	UF : 1, UT : 4,		CONFIG : 'N U T, 0, 0, 0',
	X =  145.000  mm,	Y =  154.000  mm,	Z =   15.000 mm,
	W =-180.000 deg,	P =   0.000 deg,	R =    90.000 deg
};
P[7454]{
   GP1:
	UF : 1, UT : 4,		CONFIG : 'N U T, 0, 0, 0',
	X =  145.000  mm,	Y =  154.000  mm,	Z =   -1.000 mm,
	W =-180.000 deg,	P =   0.000 deg,	R =    90.000 deg
};
P[7455]{
   GP1:
	UF : 1, UT : 4,		CONFIG : 'N U T, 0, 0, 0',
	X =  145.000  mm,	Y =  154.000  mm,	Z =   15.000 mm,
	W =-180.000 deg,	P =   0.000 deg,	R =    90.000 deg
};
P[7456]{
   GP1:
	UF : 1, UT : 4,		CONFIG : 'N U T, 0, 0, 0',
	X =  148.000  mm,	Y =  154.000  mm,	Z =   15.000 mm,
	W =-180.000 deg,	P =   0.000 deg,	R =    90.000 deg
};
P[7457]{
   GP1:
	UF : 1, UT : 4,		CONFIG : 'N U T, 0, 0, 0',
	X =  148.000  mm,	Y =  154.000  mm,	Z =   -1.000 mm,
	W =-180.000 deg,	P =   0.000 deg,	R =    90.000 deg
};
P[7458]{
   GP1:
	UF : 1, UT : 4,		CONFIG : 'N U T, 0, 0, 0',
	X =  148.000  mm,	Y =  154.000  mm,	Z =   15.000 mm,
	W =-180.000 deg,	P =   0.000 deg,	R =    90.000 deg
};
P[7459]{
   GP1:
	UF : 1, UT : 4,		CONFIG : 'N U T, 0, 0, 0',
	X =  151.000  mm,	Y =  154.000  mm,	Z =   15.000 mm,
	W =-180.000 deg,	P =   0.000 deg,	R =    90.000 deg
};
P[7460]{
   GP1:
	UF : 1, UT : 4,		CONFIG : 'N U T, 0, 0, 0',
	X =  151.000  mm,	Y =  154.000  mm,	Z =   -1.000 mm,
	W =-180.000 deg,	P =   0.000 deg,	R =    90.000 deg
};
P[7461]{
   GP1:
	UF : 1, UT : 4,		CONFIG : 'N U T, 0, 0, 0',
	X =  151.000  mm,	Y =  154.000  mm,	Z =   15.000 mm,
	W =-180.000 deg,	P =   0.000 deg,	R =    90.000 deg
};
P[7462]{
   GP1:
	UF : 1, UT : 4,		CONFIG : 'N U T, 0, 0, 0',
	X =  154.000  mm,	Y =  154.000  mm,	Z =   15.000 mm,
	W =-180.000 deg,	P =   0.000 deg,	R =    90.000 deg
};
P[7463]{
   GP1:
	UF : 1, UT : 4,		CONFIG : 'N U T, 0, 0, 0',
	X =  154.000  mm,	Y =  154.000  mm,	Z =   -1.000 mm,
	W =-180.000 deg,	P =   0.000 deg,	R =    90.000 deg
};
P[7464]{
   GP1:
	UF : 1, UT : 4,		CONFIG : 'N U T, 0, 0, 0',
	X =  154.000  mm,	Y =  154.000  mm,	Z =   15.000 mm,
	W =-180.000 deg,	P =   0.000 deg,	R =    90.000 deg
};
P[7474]{
   GP1:
	UF : 1, UT : 4,		CONFIG : 'N U T, 0, 0, 0',
	X =  25.000  mm,	Y =  157.000  mm,	Z =   15.000 mm,
	W =-180.000 deg,	P =   0.000 deg,	R =    90.000 deg
};
P[7475]{
   GP1:
	UF : 1, UT : 4,		CONFIG : 'N U T, 0, 0, 0',
	X =  25.000  mm,	Y =  157.000  mm,	Z =   -1.000 mm,
	W =-180.000 deg,	P =   0.000 deg,	R =    90.000 deg
};
P[7476]{
   GP1:
	UF : 1, UT : 4,		CONFIG : 'N U T, 0, 0, 0',
	X =  25.000  mm,	Y =  157.000  mm,	Z =   15.000 mm,
	W =-180.000 deg,	P =   0.000 deg,	R =    90.000 deg
};
P[7477]{
   GP1:
	UF : 1, UT : 4,		CONFIG : 'N U T, 0, 0, 0',
	X =  28.000  mm,	Y =  157.000  mm,	Z =   15.000 mm,
	W =-180.000 deg,	P =   0.000 deg,	R =    90.000 deg
};
P[7478]{
   GP1:
	UF : 1, UT : 4,		CONFIG : 'N U T, 0, 0, 0',
	X =  28.000  mm,	Y =  157.000  mm,	Z =   -1.000 mm,
	W =-180.000 deg,	P =   0.000 deg,	R =    90.000 deg
};
P[7479]{
   GP1:
	UF : 1, UT : 4,		CONFIG : 'N U T, 0, 0, 0',
	X =  28.000  mm,	Y =  157.000  mm,	Z =   15.000 mm,
	W =-180.000 deg,	P =   0.000 deg,	R =    90.000 deg
};
P[7480]{
   GP1:
	UF : 1, UT : 4,		CONFIG : 'N U T, 0, 0, 0',
	X =  31.000  mm,	Y =  157.000  mm,	Z =   15.000 mm,
	W =-180.000 deg,	P =   0.000 deg,	R =    90.000 deg
};
P[7481]{
   GP1:
	UF : 1, UT : 4,		CONFIG : 'N U T, 0, 0, 0',
	X =  31.000  mm,	Y =  157.000  mm,	Z =   -1.000 mm,
	W =-180.000 deg,	P =   0.000 deg,	R =    90.000 deg
};
P[7482]{
   GP1:
	UF : 1, UT : 4,		CONFIG : 'N U T, 0, 0, 0',
	X =  31.000  mm,	Y =  157.000  mm,	Z =   15.000 mm,
	W =-180.000 deg,	P =   0.000 deg,	R =    90.000 deg
};
P[7483]{
   GP1:
	UF : 1, UT : 4,		CONFIG : 'N U T, 0, 0, 0',
	X =  34.000  mm,	Y =  157.000  mm,	Z =   15.000 mm,
	W =-180.000 deg,	P =   0.000 deg,	R =    90.000 deg
};
P[7484]{
   GP1:
	UF : 1, UT : 4,		CONFIG : 'N U T, 0, 0, 0',
	X =  34.000  mm,	Y =  157.000  mm,	Z =   -1.000 mm,
	W =-180.000 deg,	P =   0.000 deg,	R =    90.000 deg
};
P[7485]{
   GP1:
	UF : 1, UT : 4,		CONFIG : 'N U T, 0, 0, 0',
	X =  34.000  mm,	Y =  157.000  mm,	Z =   15.000 mm,
	W =-180.000 deg,	P =   0.000 deg,	R =    90.000 deg
};
P[7486]{
   GP1:
	UF : 1, UT : 4,		CONFIG : 'N U T, 0, 0, 0',
	X =  37.000  mm,	Y =  157.000  mm,	Z =   15.000 mm,
	W =-180.000 deg,	P =   0.000 deg,	R =    90.000 deg
};
P[7487]{
   GP1:
	UF : 1, UT : 4,		CONFIG : 'N U T, 0, 0, 0',
	X =  37.000  mm,	Y =  157.000  mm,	Z =   -1.000 mm,
	W =-180.000 deg,	P =   0.000 deg,	R =    90.000 deg
};
P[7488]{
   GP1:
	UF : 1, UT : 4,		CONFIG : 'N U T, 0, 0, 0',
	X =  37.000  mm,	Y =  157.000  mm,	Z =   15.000 mm,
	W =-180.000 deg,	P =   0.000 deg,	R =    90.000 deg
};
P[7489]{
   GP1:
	UF : 1, UT : 4,		CONFIG : 'N U T, 0, 0, 0',
	X =  40.000  mm,	Y =  157.000  mm,	Z =   15.000 mm,
	W =-180.000 deg,	P =   0.000 deg,	R =    90.000 deg
};
P[7490]{
   GP1:
	UF : 1, UT : 4,		CONFIG : 'N U T, 0, 0, 0',
	X =  40.000  mm,	Y =  157.000  mm,	Z =   -1.000 mm,
	W =-180.000 deg,	P =   0.000 deg,	R =    90.000 deg
};
P[7491]{
   GP1:
	UF : 1, UT : 4,		CONFIG : 'N U T, 0, 0, 0',
	X =  40.000  mm,	Y =  157.000  mm,	Z =   15.000 mm,
	W =-180.000 deg,	P =   0.000 deg,	R =    90.000 deg
};
P[7492]{
   GP1:
	UF : 1, UT : 4,		CONFIG : 'N U T, 0, 0, 0',
	X =  43.000  mm,	Y =  157.000  mm,	Z =   15.000 mm,
	W =-180.000 deg,	P =   0.000 deg,	R =    90.000 deg
};
P[7493]{
   GP1:
	UF : 1, UT : 4,		CONFIG : 'N U T, 0, 0, 0',
	X =  43.000  mm,	Y =  157.000  mm,	Z =   -1.000 mm,
	W =-180.000 deg,	P =   0.000 deg,	R =    90.000 deg
};
P[7494]{
   GP1:
	UF : 1, UT : 4,		CONFIG : 'N U T, 0, 0, 0',
	X =  43.000  mm,	Y =  157.000  mm,	Z =   15.000 mm,
	W =-180.000 deg,	P =   0.000 deg,	R =    90.000 deg
};
P[7495]{
   GP1:
	UF : 1, UT : 4,		CONFIG : 'N U T, 0, 0, 0',
	X =  46.000  mm,	Y =  157.000  mm,	Z =   15.000 mm,
	W =-180.000 deg,	P =   0.000 deg,	R =    90.000 deg
};
P[7496]{
   GP1:
	UF : 1, UT : 4,		CONFIG : 'N U T, 0, 0, 0',
	X =  46.000  mm,	Y =  157.000  mm,	Z =   -1.000 mm,
	W =-180.000 deg,	P =   0.000 deg,	R =    90.000 deg
};
P[7497]{
   GP1:
	UF : 1, UT : 4,		CONFIG : 'N U T, 0, 0, 0',
	X =  46.000  mm,	Y =  157.000  mm,	Z =   15.000 mm,
	W =-180.000 deg,	P =   0.000 deg,	R =    90.000 deg
};
P[7498]{
   GP1:
	UF : 1, UT : 4,		CONFIG : 'N U T, 0, 0, 0',
	X =  49.000  mm,	Y =  157.000  mm,	Z =   15.000 mm,
	W =-180.000 deg,	P =   0.000 deg,	R =    90.000 deg
};
P[7499]{
   GP1:
	UF : 1, UT : 4,		CONFIG : 'N U T, 0, 0, 0',
	X =  49.000  mm,	Y =  157.000  mm,	Z =   -1.000 mm,
	W =-180.000 deg,	P =   0.000 deg,	R =    90.000 deg
};
P[7500]{
   GP1:
	UF : 1, UT : 4,		CONFIG : 'N U T, 0, 0, 0',
	X =  49.000  mm,	Y =  157.000  mm,	Z =   15.000 mm,
	W =-180.000 deg,	P =   0.000 deg,	R =    90.000 deg
};
P[7501]{
   GP1:
	UF : 1, UT : 4,		CONFIG : 'N U T, 0, 0, 0',
	X =  52.000  mm,	Y =  157.000  mm,	Z =   15.000 mm,
	W =-180.000 deg,	P =   0.000 deg,	R =    90.000 deg
};
P[7502]{
   GP1:
	UF : 1, UT : 4,		CONFIG : 'N U T, 0, 0, 0',
	X =  52.000  mm,	Y =  157.000  mm,	Z =   -1.000 mm,
	W =-180.000 deg,	P =   0.000 deg,	R =    90.000 deg
};
P[7503]{
   GP1:
	UF : 1, UT : 4,		CONFIG : 'N U T, 0, 0, 0',
	X =  52.000  mm,	Y =  157.000  mm,	Z =   15.000 mm,
	W =-180.000 deg,	P =   0.000 deg,	R =    90.000 deg
};
P[7504]{
   GP1:
	UF : 1, UT : 4,		CONFIG : 'N U T, 0, 0, 0',
	X =  55.000  mm,	Y =  157.000  mm,	Z =   15.000 mm,
	W =-180.000 deg,	P =   0.000 deg,	R =    90.000 deg
};
P[7505]{
   GP1:
	UF : 1, UT : 4,		CONFIG : 'N U T, 0, 0, 0',
	X =  55.000  mm,	Y =  157.000  mm,	Z =   -1.000 mm,
	W =-180.000 deg,	P =   0.000 deg,	R =    90.000 deg
};
P[7506]{
   GP1:
	UF : 1, UT : 4,		CONFIG : 'N U T, 0, 0, 0',
	X =  55.000  mm,	Y =  157.000  mm,	Z =   15.000 mm,
	W =-180.000 deg,	P =   0.000 deg,	R =    90.000 deg
};
P[7507]{
   GP1:
	UF : 1, UT : 4,		CONFIG : 'N U T, 0, 0, 0',
	X =  58.000  mm,	Y =  157.000  mm,	Z =   15.000 mm,
	W =-180.000 deg,	P =   0.000 deg,	R =    90.000 deg
};
P[7508]{
   GP1:
	UF : 1, UT : 4,		CONFIG : 'N U T, 0, 0, 0',
	X =  58.000  mm,	Y =  157.000  mm,	Z =   -1.000 mm,
	W =-180.000 deg,	P =   0.000 deg,	R =    90.000 deg
};
P[7509]{
   GP1:
	UF : 1, UT : 4,		CONFIG : 'N U T, 0, 0, 0',
	X =  58.000  mm,	Y =  157.000  mm,	Z =   15.000 mm,
	W =-180.000 deg,	P =   0.000 deg,	R =    90.000 deg
};
P[7516]{
   GP1:
	UF : 1, UT : 4,		CONFIG : 'N U T, 0, 0, 0',
	X =  109.000  mm,	Y =  157.000  mm,	Z =   15.000 mm,
	W =-180.000 deg,	P =   0.000 deg,	R =    90.000 deg
};
P[7517]{
   GP1:
	UF : 1, UT : 4,		CONFIG : 'N U T, 0, 0, 0',
	X =  109.000  mm,	Y =  157.000  mm,	Z =   -1.000 mm,
	W =-180.000 deg,	P =   0.000 deg,	R =    90.000 deg
};
P[7518]{
   GP1:
	UF : 1, UT : 4,		CONFIG : 'N U T, 0, 0, 0',
	X =  109.000  mm,	Y =  157.000  mm,	Z =   15.000 mm,
	W =-180.000 deg,	P =   0.000 deg,	R =    90.000 deg
};
P[7549]{
   GP1:
	UF : 1, UT : 4,		CONFIG : 'N U T, 0, 0, 0',
	X =  142.000  mm,	Y =  157.000  mm,	Z =   15.000 mm,
	W =-180.000 deg,	P =   0.000 deg,	R =    90.000 deg
};
P[7550]{
   GP1:
	UF : 1, UT : 4,		CONFIG : 'N U T, 0, 0, 0',
	X =  142.000  mm,	Y =  157.000  mm,	Z =   -1.000 mm,
	W =-180.000 deg,	P =   0.000 deg,	R =    90.000 deg
};
P[7551]{
   GP1:
	UF : 1, UT : 4,		CONFIG : 'N U T, 0, 0, 0',
	X =  142.000  mm,	Y =  157.000  mm,	Z =   15.000 mm,
	W =-180.000 deg,	P =   0.000 deg,	R =    90.000 deg
};
P[7552]{
   GP1:
	UF : 1, UT : 4,		CONFIG : 'N U T, 0, 0, 0',
	X =  145.000  mm,	Y =  157.000  mm,	Z =   15.000 mm,
	W =-180.000 deg,	P =   0.000 deg,	R =    90.000 deg
};
P[7553]{
   GP1:
	UF : 1, UT : 4,		CONFIG : 'N U T, 0, 0, 0',
	X =  145.000  mm,	Y =  157.000  mm,	Z =   -1.000 mm,
	W =-180.000 deg,	P =   0.000 deg,	R =    90.000 deg
};
P[7554]{
   GP1:
	UF : 1, UT : 4,		CONFIG : 'N U T, 0, 0, 0',
	X =  145.000  mm,	Y =  157.000  mm,	Z =   15.000 mm,
	W =-180.000 deg,	P =   0.000 deg,	R =    90.000 deg
};
P[7555]{
   GP1:
	UF : 1, UT : 4,		CONFIG : 'N U T, 0, 0, 0',
	X =  148.000  mm,	Y =  157.000  mm,	Z =   15.000 mm,
	W =-180.000 deg,	P =   0.000 deg,	R =    90.000 deg
};
P[7556]{
   GP1:
	UF : 1, UT : 4,		CONFIG : 'N U T, 0, 0, 0',
	X =  148.000  mm,	Y =  157.000  mm,	Z =   -1.000 mm,
	W =-180.000 deg,	P =   0.000 deg,	R =    90.000 deg
};
P[7557]{
   GP1:
	UF : 1, UT : 4,		CONFIG : 'N U T, 0, 0, 0',
	X =  148.000  mm,	Y =  157.000  mm,	Z =   15.000 mm,
	W =-180.000 deg,	P =   0.000 deg,	R =    90.000 deg
};
P[7558]{
   GP1:
	UF : 1, UT : 4,		CONFIG : 'N U T, 0, 0, 0',
	X =  151.000  mm,	Y =  157.000  mm,	Z =   15.000 mm,
	W =-180.000 deg,	P =   0.000 deg,	R =    90.000 deg
};
P[7559]{
   GP1:
	UF : 1, UT : 4,		CONFIG : 'N U T, 0, 0, 0',
	X =  151.000  mm,	Y =  157.000  mm,	Z =   -1.000 mm,
	W =-180.000 deg,	P =   0.000 deg,	R =    90.000 deg
};
P[7560]{
   GP1:
	UF : 1, UT : 4,		CONFIG : 'N U T, 0, 0, 0',
	X =  151.000  mm,	Y =  157.000  mm,	Z =   15.000 mm,
	W =-180.000 deg,	P =   0.000 deg,	R =    90.000 deg
};
P[7561]{
   GP1:
	UF : 1, UT : 4,		CONFIG : 'N U T, 0, 0, 0',
	X =  154.000  mm,	Y =  157.000  mm,	Z =   15.000 mm,
	W =-180.000 deg,	P =   0.000 deg,	R =    90.000 deg
};
P[7562]{
   GP1:
	UF : 1, UT : 4,		CONFIG : 'N U T, 0, 0, 0',
	X =  154.000  mm,	Y =  157.000  mm,	Z =   -1.000 mm,
	W =-180.000 deg,	P =   0.000 deg,	R =    90.000 deg
};
P[7563]{
   GP1:
	UF : 1, UT : 4,		CONFIG : 'N U T, 0, 0, 0',
	X =  154.000  mm,	Y =  157.000  mm,	Z =   15.000 mm,
	W =-180.000 deg,	P =   0.000 deg,	R =    90.000 deg
};
P[7615]{
   GP1:
	UF : 1, UT : 4,		CONFIG : 'N U T, 0, 0, 0',
	X =  109.000  mm,	Y =  160.000  mm,	Z =   15.000 mm,
	W =-180.000 deg,	P =   0.000 deg,	R =    90.000 deg
};
P[7616]{
   GP1:
	UF : 1, UT : 4,		CONFIG : 'N U T, 0, 0, 0',
	X =  109.000  mm,	Y =  160.000  mm,	Z =   -1.000 mm,
	W =-180.000 deg,	P =   0.000 deg,	R =    90.000 deg
};
P[7617]{
   GP1:
	UF : 1, UT : 4,		CONFIG : 'N U T, 0, 0, 0',
	X =  109.000  mm,	Y =  160.000  mm,	Z =   15.000 mm,
	W =-180.000 deg,	P =   0.000 deg,	R =    90.000 deg
};
P[7618]{
   GP1:
	UF : 1, UT : 4,		CONFIG : 'N U T, 0, 0, 0',
	X =  112.000  mm,	Y =  160.000  mm,	Z =   15.000 mm,
	W =-180.000 deg,	P =   0.000 deg,	R =    90.000 deg
};
P[7619]{
   GP1:
	UF : 1, UT : 4,		CONFIG : 'N U T, 0, 0, 0',
	X =  112.000  mm,	Y =  160.000  mm,	Z =   -1.000 mm,
	W =-180.000 deg,	P =   0.000 deg,	R =    90.000 deg
};
P[7620]{
   GP1:
	UF : 1, UT : 4,		CONFIG : 'N U T, 0, 0, 0',
	X =  112.000  mm,	Y =  160.000  mm,	Z =   15.000 mm,
	W =-180.000 deg,	P =   0.000 deg,	R =    90.000 deg
};
P[7651]{
   GP1:
	UF : 1, UT : 4,		CONFIG : 'N U T, 0, 0, 0',
	X =  145.000  mm,	Y =  160.000  mm,	Z =   15.000 mm,
	W =-180.000 deg,	P =   0.000 deg,	R =    90.000 deg
};
P[7652]{
   GP1:
	UF : 1, UT : 4,		CONFIG : 'N U T, 0, 0, 0',
	X =  145.000  mm,	Y =  160.000  mm,	Z =   -1.000 mm,
	W =-180.000 deg,	P =   0.000 deg,	R =    90.000 deg
};
P[7653]{
   GP1:
	UF : 1, UT : 4,		CONFIG : 'N U T, 0, 0, 0',
	X =  145.000  mm,	Y =  160.000  mm,	Z =   15.000 mm,
	W =-180.000 deg,	P =   0.000 deg,	R =    90.000 deg
};
P[7654]{
   GP1:
	UF : 1, UT : 4,		CONFIG : 'N U T, 0, 0, 0',
	X =  148.000  mm,	Y =  160.000  mm,	Z =   15.000 mm,
	W =-180.000 deg,	P =   0.000 deg,	R =    90.000 deg
};
P[7655]{
   GP1:
	UF : 1, UT : 4,		CONFIG : 'N U T, 0, 0, 0',
	X =  148.000  mm,	Y =  160.000  mm,	Z =   -1.000 mm,
	W =-180.000 deg,	P =   0.000 deg,	R =    90.000 deg
};
P[7656]{
   GP1:
	UF : 1, UT : 4,		CONFIG : 'N U T, 0, 0, 0',
	X =  148.000  mm,	Y =  160.000  mm,	Z =   15.000 mm,
	W =-180.000 deg,	P =   0.000 deg,	R =    90.000 deg
};
P[7663]{
   GP1:
	UF : 1, UT : 4,		CONFIG : 'N U T, 0, 0, 0',
	X =  22.000  mm,	Y =  163.000  mm,	Z =   15.000 mm,
	W =-180.000 deg,	P =   0.000 deg,	R =    90.000 deg
};
P[7664]{
   GP1:
	UF : 1, UT : 4,		CONFIG : 'N U T, 0, 0, 0',
	X =  22.000  mm,	Y =  163.000  mm,	Z =   -1.000 mm,
	W =-180.000 deg,	P =   0.000 deg,	R =    90.000 deg
};
P[7665]{
   GP1:
	UF : 1, UT : 4,		CONFIG : 'N U T, 0, 0, 0',
	X =  22.000  mm,	Y =  163.000  mm,	Z =   15.000 mm,
	W =-180.000 deg,	P =   0.000 deg,	R =    90.000 deg
};
P[7708]{
   GP1:
	UF : 1, UT : 4,		CONFIG : 'N U T, 0, 0, 0',
	X =  109.000  mm,	Y =  163.000  mm,	Z =   15.000 mm,
	W =-180.000 deg,	P =   0.000 deg,	R =    90.000 deg
};
P[7709]{
   GP1:
	UF : 1, UT : 4,		CONFIG : 'N U T, 0, 0, 0',
	X =  109.000  mm,	Y =  163.000  mm,	Z =   -1.000 mm,
	W =-180.000 deg,	P =   0.000 deg,	R =    90.000 deg
};
P[7710]{
   GP1:
	UF : 1, UT : 4,		CONFIG : 'N U T, 0, 0, 0',
	X =  109.000  mm,	Y =  163.000  mm,	Z =   15.000 mm,
	W =-180.000 deg,	P =   0.000 deg,	R =    90.000 deg
};
P[7711]{
   GP1:
	UF : 1, UT : 4,		CONFIG : 'N U T, 0, 0, 0',
	X =  112.000  mm,	Y =  163.000  mm,	Z =   15.000 mm,
	W =-180.000 deg,	P =   0.000 deg,	R =    90.000 deg
};
P[7712]{
   GP1:
	UF : 1, UT : 4,		CONFIG : 'N U T, 0, 0, 0',
	X =  112.000  mm,	Y =  163.000  mm,	Z =   -1.000 mm,
	W =-180.000 deg,	P =   0.000 deg,	R =    90.000 deg
};
P[7713]{
   GP1:
	UF : 1, UT : 4,		CONFIG : 'N U T, 0, 0, 0',
	X =  112.000  mm,	Y =  163.000  mm,	Z =   15.000 mm,
	W =-180.000 deg,	P =   0.000 deg,	R =    90.000 deg
};
P[7720]{
   GP1:
	UF : 1, UT : 4,		CONFIG : 'N U T, 0, 0, 0',
	X =  121.000  mm,	Y =  163.000  mm,	Z =   15.000 mm,
	W =-180.000 deg,	P =   0.000 deg,	R =    90.000 deg
};
P[7721]{
   GP1:
	UF : 1, UT : 4,		CONFIG : 'N U T, 0, 0, 0',
	X =  121.000  mm,	Y =  163.000  mm,	Z =   -1.000 mm,
	W =-180.000 deg,	P =   0.000 deg,	R =    90.000 deg
};
P[7722]{
   GP1:
	UF : 1, UT : 4,		CONFIG : 'N U T, 0, 0, 0',
	X =  121.000  mm,	Y =  163.000  mm,	Z =   15.000 mm,
	W =-180.000 deg,	P =   0.000 deg,	R =    90.000 deg
};
P[7723]{
   GP1:
	UF : 1, UT : 4,		CONFIG : 'N U T, 0, 0, 0',
	X =  124.000  mm,	Y =  163.000  mm,	Z =   15.000 mm,
	W =-180.000 deg,	P =   0.000 deg,	R =    90.000 deg
};
P[7724]{
   GP1:
	UF : 1, UT : 4,		CONFIG : 'N U T, 0, 0, 0',
	X =  124.000  mm,	Y =  163.000  mm,	Z =   -1.000 mm,
	W =-180.000 deg,	P =   0.000 deg,	R =    90.000 deg
};
P[7725]{
   GP1:
	UF : 1, UT : 4,		CONFIG : 'N U T, 0, 0, 0',
	X =  124.000  mm,	Y =  163.000  mm,	Z =   15.000 mm,
	W =-180.000 deg,	P =   0.000 deg,	R =    90.000 deg
};
P[7726]{
   GP1:
	UF : 1, UT : 4,		CONFIG : 'N U T, 0, 0, 0',
	X =  127.000  mm,	Y =  163.000  mm,	Z =   15.000 mm,
	W =-180.000 deg,	P =   0.000 deg,	R =    90.000 deg
};
P[7727]{
   GP1:
	UF : 1, UT : 4,		CONFIG : 'N U T, 0, 0, 0',
	X =  127.000  mm,	Y =  163.000  mm,	Z =   -1.000 mm,
	W =-180.000 deg,	P =   0.000 deg,	R =    90.000 deg
};
P[7728]{
   GP1:
	UF : 1, UT : 4,		CONFIG : 'N U T, 0, 0, 0',
	X =  127.000  mm,	Y =  163.000  mm,	Z =   15.000 mm,
	W =-180.000 deg,	P =   0.000 deg,	R =    90.000 deg
};
P[7729]{
   GP1:
	UF : 1, UT : 4,		CONFIG : 'N U T, 0, 0, 0',
	X =  130.000  mm,	Y =  163.000  mm,	Z =   15.000 mm,
	W =-180.000 deg,	P =   0.000 deg,	R =    90.000 deg
};
P[7730]{
   GP1:
	UF : 1, UT : 4,		CONFIG : 'N U T, 0, 0, 0',
	X =  130.000  mm,	Y =  163.000  mm,	Z =   -1.000 mm,
	W =-180.000 deg,	P =   0.000 deg,	R =    90.000 deg
};
P[7731]{
   GP1:
	UF : 1, UT : 4,		CONFIG : 'N U T, 0, 0, 0',
	X =  130.000  mm,	Y =  163.000  mm,	Z =   15.000 mm,
	W =-180.000 deg,	P =   0.000 deg,	R =    90.000 deg
};
P[7732]{
   GP1:
	UF : 1, UT : 4,		CONFIG : 'N U T, 0, 0, 0',
	X =  133.000  mm,	Y =  163.000  mm,	Z =   15.000 mm,
	W =-180.000 deg,	P =   0.000 deg,	R =    90.000 deg
};
P[7733]{
   GP1:
	UF : 1, UT : 4,		CONFIG : 'N U T, 0, 0, 0',
	X =  133.000  mm,	Y =  163.000  mm,	Z =   -1.000 mm,
	W =-180.000 deg,	P =   0.000 deg,	R =    90.000 deg
};
P[7734]{
   GP1:
	UF : 1, UT : 4,		CONFIG : 'N U T, 0, 0, 0',
	X =  133.000  mm,	Y =  163.000  mm,	Z =   15.000 mm,
	W =-180.000 deg,	P =   0.000 deg,	R =    90.000 deg
};
P[7735]{
   GP1:
	UF : 1, UT : 4,		CONFIG : 'N U T, 0, 0, 0',
	X =  136.000  mm,	Y =  163.000  mm,	Z =   15.000 mm,
	W =-180.000 deg,	P =   0.000 deg,	R =    90.000 deg
};
P[7736]{
   GP1:
	UF : 1, UT : 4,		CONFIG : 'N U T, 0, 0, 0',
	X =  136.000  mm,	Y =  163.000  mm,	Z =   -1.000 mm,
	W =-180.000 deg,	P =   0.000 deg,	R =    90.000 deg
};
P[7737]{
   GP1:
	UF : 1, UT : 4,		CONFIG : 'N U T, 0, 0, 0',
	X =  136.000  mm,	Y =  163.000  mm,	Z =   15.000 mm,
	W =-180.000 deg,	P =   0.000 deg,	R =    90.000 deg
};
P[7738]{
   GP1:
	UF : 1, UT : 4,		CONFIG : 'N U T, 0, 0, 0',
	X =  139.000  mm,	Y =  163.000  mm,	Z =   15.000 mm,
	W =-180.000 deg,	P =   0.000 deg,	R =    90.000 deg
};
P[7739]{
   GP1:
	UF : 1, UT : 4,		CONFIG : 'N U T, 0, 0, 0',
	X =  139.000  mm,	Y =  163.000  mm,	Z =   -1.000 mm,
	W =-180.000 deg,	P =   0.000 deg,	R =    90.000 deg
};
P[7740]{
   GP1:
	UF : 1, UT : 4,		CONFIG : 'N U T, 0, 0, 0',
	X =  139.000  mm,	Y =  163.000  mm,	Z =   15.000 mm,
	W =-180.000 deg,	P =   0.000 deg,	R =    90.000 deg
};
P[7741]{
   GP1:
	UF : 1, UT : 4,		CONFIG : 'N U T, 0, 0, 0',
	X =  142.000  mm,	Y =  163.000  mm,	Z =   15.000 mm,
	W =-180.000 deg,	P =   0.000 deg,	R =    90.000 deg
};
P[7742]{
   GP1:
	UF : 1, UT : 4,		CONFIG : 'N U T, 0, 0, 0',
	X =  142.000  mm,	Y =  163.000  mm,	Z =   -1.000 mm,
	W =-180.000 deg,	P =   0.000 deg,	R =    90.000 deg
};
P[7743]{
   GP1:
	UF : 1, UT : 4,		CONFIG : 'N U T, 0, 0, 0',
	X =  142.000  mm,	Y =  163.000  mm,	Z =   15.000 mm,
	W =-180.000 deg,	P =   0.000 deg,	R =    90.000 deg
};
P[7744]{
   GP1:
	UF : 1, UT : 4,		CONFIG : 'N U T, 0, 0, 0',
	X =  145.000  mm,	Y =  163.000  mm,	Z =   15.000 mm,
	W =-180.000 deg,	P =   0.000 deg,	R =    90.000 deg
};
P[7745]{
   GP1:
	UF : 1, UT : 4,		CONFIG : 'N U T, 0, 0, 0',
	X =  145.000  mm,	Y =  163.000  mm,	Z =   -1.000 mm,
	W =-180.000 deg,	P =   0.000 deg,	R =    90.000 deg
};
P[7746]{
   GP1:
	UF : 1, UT : 4,		CONFIG : 'N U T, 0, 0, 0',
	X =  145.000  mm,	Y =  163.000  mm,	Z =   15.000 mm,
	W =-180.000 deg,	P =   0.000 deg,	R =    90.000 deg
};
P[7747]{
   GP1:
	UF : 1, UT : 4,		CONFIG : 'N U T, 0, 0, 0',
	X =  148.000  mm,	Y =  163.000  mm,	Z =   15.000 mm,
	W =-180.000 deg,	P =   0.000 deg,	R =    90.000 deg
};
P[7748]{
   GP1:
	UF : 1, UT : 4,		CONFIG : 'N U T, 0, 0, 0',
	X =  148.000  mm,	Y =  163.000  mm,	Z =   -1.000 mm,
	W =-180.000 deg,	P =   0.000 deg,	R =    90.000 deg
};
P[7749]{
   GP1:
	UF : 1, UT : 4,		CONFIG : 'N U T, 0, 0, 0',
	X =  148.000  mm,	Y =  163.000  mm,	Z =   15.000 mm,
	W =-180.000 deg,	P =   0.000 deg,	R =    90.000 deg
};
P[7780]{
   GP1:
	UF : 1, UT : 4,		CONFIG : 'N U T, 0, 0, 0',
	X =  49.000  mm,	Y =  166.000  mm,	Z =   15.000 mm,
	W =-180.000 deg,	P =   0.000 deg,	R =    90.000 deg
};
P[7781]{
   GP1:
	UF : 1, UT : 4,		CONFIG : 'N U T, 0, 0, 0',
	X =  49.000  mm,	Y =  166.000  mm,	Z =   -1.000 mm,
	W =-180.000 deg,	P =   0.000 deg,	R =    90.000 deg
};
P[7782]{
   GP1:
	UF : 1, UT : 4,		CONFIG : 'N U T, 0, 0, 0',
	X =  49.000  mm,	Y =  166.000  mm,	Z =   15.000 mm,
	W =-180.000 deg,	P =   0.000 deg,	R =    90.000 deg
};
P[7795]{
   GP1:
	UF : 1, UT : 4,		CONFIG : 'N U T, 0, 0, 0',
	X =  109.000  mm,	Y =  166.000  mm,	Z =   15.000 mm,
	W =-180.000 deg,	P =   0.000 deg,	R =    90.000 deg
};
P[7796]{
   GP1:
	UF : 1, UT : 4,		CONFIG : 'N U T, 0, 0, 0',
	X =  109.000  mm,	Y =  166.000  mm,	Z =   -1.000 mm,
	W =-180.000 deg,	P =   0.000 deg,	R =    90.000 deg
};
P[7797]{
   GP1:
	UF : 1, UT : 4,		CONFIG : 'N U T, 0, 0, 0',
	X =  109.000  mm,	Y =  166.000  mm,	Z =   15.000 mm,
	W =-180.000 deg,	P =   0.000 deg,	R =    90.000 deg
};
P[7798]{
   GP1:
	UF : 1, UT : 4,		CONFIG : 'N U T, 0, 0, 0',
	X =  112.000  mm,	Y =  166.000  mm,	Z =   15.000 mm,
	W =-180.000 deg,	P =   0.000 deg,	R =    90.000 deg
};
P[7799]{
   GP1:
	UF : 1, UT : 4,		CONFIG : 'N U T, 0, 0, 0',
	X =  112.000  mm,	Y =  166.000  mm,	Z =   -1.000 mm,
	W =-180.000 deg,	P =   0.000 deg,	R =    90.000 deg
};
P[7800]{
   GP1:
	UF : 1, UT : 4,		CONFIG : 'N U T, 0, 0, 0',
	X =  112.000  mm,	Y =  166.000  mm,	Z =   15.000 mm,
	W =-180.000 deg,	P =   0.000 deg,	R =    90.000 deg
};
P[7813]{
   GP1:
	UF : 1, UT : 4,		CONFIG : 'N U T, 0, 0, 0',
	X =  127.000  mm,	Y =  166.000  mm,	Z =   15.000 mm,
	W =-180.000 deg,	P =   0.000 deg,	R =    90.000 deg
};
P[7814]{
   GP1:
	UF : 1, UT : 4,		CONFIG : 'N U T, 0, 0, 0',
	X =  127.000  mm,	Y =  166.000  mm,	Z =   -1.000 mm,
	W =-180.000 deg,	P =   0.000 deg,	R =    90.000 deg
};
P[7815]{
   GP1:
	UF : 1, UT : 4,		CONFIG : 'N U T, 0, 0, 0',
	X =  127.000  mm,	Y =  166.000  mm,	Z =   15.000 mm,
	W =-180.000 deg,	P =   0.000 deg,	R =    90.000 deg
};
P[7816]{
   GP1:
	UF : 1, UT : 4,		CONFIG : 'N U T, 0, 0, 0',
	X =  130.000  mm,	Y =  166.000  mm,	Z =   15.000 mm,
	W =-180.000 deg,	P =   0.000 deg,	R =    90.000 deg
};
P[7817]{
   GP1:
	UF : 1, UT : 4,		CONFIG : 'N U T, 0, 0, 0',
	X =  130.000  mm,	Y =  166.000  mm,	Z =   -1.000 mm,
	W =-180.000 deg,	P =   0.000 deg,	R =    90.000 deg
};
P[7818]{
   GP1:
	UF : 1, UT : 4,		CONFIG : 'N U T, 0, 0, 0',
	X =  130.000  mm,	Y =  166.000  mm,	Z =   15.000 mm,
	W =-180.000 deg,	P =   0.000 deg,	R =    90.000 deg
};
P[7819]{
   GP1:
	UF : 1, UT : 4,		CONFIG : 'N U T, 0, 0, 0',
	X =  133.000  mm,	Y =  166.000  mm,	Z =   15.000 mm,
	W =-180.000 deg,	P =   0.000 deg,	R =    90.000 deg
};
P[7820]{
   GP1:
	UF : 1, UT : 4,		CONFIG : 'N U T, 0, 0, 0',
	X =  133.000  mm,	Y =  166.000  mm,	Z =   -1.000 mm,
	W =-180.000 deg,	P =   0.000 deg,	R =    90.000 deg
};
P[7821]{
   GP1:
	UF : 1, UT : 4,		CONFIG : 'N U T, 0, 0, 0',
	X =  133.000  mm,	Y =  166.000  mm,	Z =   15.000 mm,
	W =-180.000 deg,	P =   0.000 deg,	R =    90.000 deg
};
P[7822]{
   GP1:
	UF : 1, UT : 4,		CONFIG : 'N U T, 0, 0, 0',
	X =  136.000  mm,	Y =  166.000  mm,	Z =   15.000 mm,
	W =-180.000 deg,	P =   0.000 deg,	R =    90.000 deg
};
P[7823]{
   GP1:
	UF : 1, UT : 4,		CONFIG : 'N U T, 0, 0, 0',
	X =  136.000  mm,	Y =  166.000  mm,	Z =   -1.000 mm,
	W =-180.000 deg,	P =   0.000 deg,	R =    90.000 deg
};
P[7824]{
   GP1:
	UF : 1, UT : 4,		CONFIG : 'N U T, 0, 0, 0',
	X =  136.000  mm,	Y =  166.000  mm,	Z =   15.000 mm,
	W =-180.000 deg,	P =   0.000 deg,	R =    90.000 deg
};
P[7825]{
   GP1:
	UF : 1, UT : 4,		CONFIG : 'N U T, 0, 0, 0',
	X =  139.000  mm,	Y =  166.000  mm,	Z =   15.000 mm,
	W =-180.000 deg,	P =   0.000 deg,	R =    90.000 deg
};
P[7826]{
   GP1:
	UF : 1, UT : 4,		CONFIG : 'N U T, 0, 0, 0',
	X =  139.000  mm,	Y =  166.000  mm,	Z =   -1.000 mm,
	W =-180.000 deg,	P =   0.000 deg,	R =    90.000 deg
};
P[7827]{
   GP1:
	UF : 1, UT : 4,		CONFIG : 'N U T, 0, 0, 0',
	X =  139.000  mm,	Y =  166.000  mm,	Z =   15.000 mm,
	W =-180.000 deg,	P =   0.000 deg,	R =    90.000 deg
};
P[7828]{
   GP1:
	UF : 1, UT : 4,		CONFIG : 'N U T, 0, 0, 0',
	X =  142.000  mm,	Y =  166.000  mm,	Z =   15.000 mm,
	W =-180.000 deg,	P =   0.000 deg,	R =    90.000 deg
};
P[7829]{
   GP1:
	UF : 1, UT : 4,		CONFIG : 'N U T, 0, 0, 0',
	X =  142.000  mm,	Y =  166.000  mm,	Z =   -1.000 mm,
	W =-180.000 deg,	P =   0.000 deg,	R =    90.000 deg
};
P[7830]{
   GP1:
	UF : 1, UT : 4,		CONFIG : 'N U T, 0, 0, 0',
	X =  142.000  mm,	Y =  166.000  mm,	Z =   15.000 mm,
	W =-180.000 deg,	P =   0.000 deg,	R =    90.000 deg
};
P[7831]{
   GP1:
	UF : 1, UT : 4,		CONFIG : 'N U T, 0, 0, 0',
	X =  145.000  mm,	Y =  166.000  mm,	Z =   15.000 mm,
	W =-180.000 deg,	P =   0.000 deg,	R =    90.000 deg
};
P[7832]{
   GP1:
	UF : 1, UT : 4,		CONFIG : 'N U T, 0, 0, 0',
	X =  145.000  mm,	Y =  166.000  mm,	Z =   -1.000 mm,
	W =-180.000 deg,	P =   0.000 deg,	R =    90.000 deg
};
P[7833]{
   GP1:
	UF : 1, UT : 4,		CONFIG : 'N U T, 0, 0, 0',
	X =  145.000  mm,	Y =  166.000  mm,	Z =   15.000 mm,
	W =-180.000 deg,	P =   0.000 deg,	R =    90.000 deg
};
P[7834]{
   GP1:
	UF : 1, UT : 4,		CONFIG : 'N U T, 0, 0, 0',
	X =  148.000  mm,	Y =  166.000  mm,	Z =   15.000 mm,
	W =-180.000 deg,	P =   0.000 deg,	R =    90.000 deg
};
P[7835]{
   GP1:
	UF : 1, UT : 4,		CONFIG : 'N U T, 0, 0, 0',
	X =  148.000  mm,	Y =  166.000  mm,	Z =   -1.000 mm,
	W =-180.000 deg,	P =   0.000 deg,	R =    90.000 deg
};
P[7836]{
   GP1:
	UF : 1, UT : 4,		CONFIG : 'N U T, 0, 0, 0',
	X =  148.000  mm,	Y =  166.000  mm,	Z =   15.000 mm,
	W =-180.000 deg,	P =   0.000 deg,	R =    90.000 deg
};
P[7846]{
   GP1:
	UF : 1, UT : 4,		CONFIG : 'N U T, 0, 0, 0',
	X =  31.000  mm,	Y =  169.000  mm,	Z =   15.000 mm,
	W =-180.000 deg,	P =   0.000 deg,	R =    90.000 deg
};
P[7847]{
   GP1:
	UF : 1, UT : 4,		CONFIG : 'N U T, 0, 0, 0',
	X =  31.000  mm,	Y =  169.000  mm,	Z =   -1.000 mm,
	W =-180.000 deg,	P =   0.000 deg,	R =    90.000 deg
};
P[7848]{
   GP1:
	UF : 1, UT : 4,		CONFIG : 'N U T, 0, 0, 0',
	X =  31.000  mm,	Y =  169.000  mm,	Z =   15.000 mm,
	W =-180.000 deg,	P =   0.000 deg,	R =    90.000 deg
};
P[7861]{
   GP1:
	UF : 1, UT : 4,		CONFIG : 'N U T, 0, 0, 0',
	X =  46.000  mm,	Y =  169.000  mm,	Z =   15.000 mm,
	W =-180.000 deg,	P =   0.000 deg,	R =    90.000 deg
};
P[7862]{
   GP1:
	UF : 1, UT : 4,		CONFIG : 'N U T, 0, 0, 0',
	X =  46.000  mm,	Y =  169.000  mm,	Z =   -1.000 mm,
	W =-180.000 deg,	P =   0.000 deg,	R =    90.000 deg
};
P[7863]{
   GP1:
	UF : 1, UT : 4,		CONFIG : 'N U T, 0, 0, 0',
	X =  46.000  mm,	Y =  169.000  mm,	Z =   15.000 mm,
	W =-180.000 deg,	P =   0.000 deg,	R =    90.000 deg
};
P[7867]{
   GP1:
	UF : 1, UT : 4,		CONFIG : 'N U T, 0, 0, 0',
	X =  52.000  mm,	Y =  169.000  mm,	Z =   15.000 mm,
	W =-180.000 deg,	P =   0.000 deg,	R =    90.000 deg
};
P[7868]{
   GP1:
	UF : 1, UT : 4,		CONFIG : 'N U T, 0, 0, 0',
	X =  52.000  mm,	Y =  169.000  mm,	Z =   -1.000 mm,
	W =-180.000 deg,	P =   0.000 deg,	R =    90.000 deg
};
P[7869]{
   GP1:
	UF : 1, UT : 4,		CONFIG : 'N U T, 0, 0, 0',
	X =  52.000  mm,	Y =  169.000  mm,	Z =   15.000 mm,
	W =-180.000 deg,	P =   0.000 deg,	R =    90.000 deg
};
P[7876]{
   GP1:
	UF : 1, UT : 4,		CONFIG : 'N U T, 0, 0, 0',
	X =  109.000  mm,	Y =  169.000  mm,	Z =   15.000 mm,
	W =-180.000 deg,	P =   0.000 deg,	R =    90.000 deg
};
P[7877]{
   GP1:
	UF : 1, UT : 4,		CONFIG : 'N U T, 0, 0, 0',
	X =  109.000  mm,	Y =  169.000  mm,	Z =   -1.000 mm,
	W =-180.000 deg,	P =   0.000 deg,	R =    90.000 deg
};
P[7878]{
   GP1:
	UF : 1, UT : 4,		CONFIG : 'N U T, 0, 0, 0',
	X =  109.000  mm,	Y =  169.000  mm,	Z =   15.000 mm,
	W =-180.000 deg,	P =   0.000 deg,	R =    90.000 deg
};
P[7879]{
   GP1:
	UF : 1, UT : 4,		CONFIG : 'N U T, 0, 0, 0',
	X =  112.000  mm,	Y =  169.000  mm,	Z =   15.000 mm,
	W =-180.000 deg,	P =   0.000 deg,	R =    90.000 deg
};
P[7880]{
   GP1:
	UF : 1, UT : 4,		CONFIG : 'N U T, 0, 0, 0',
	X =  112.000  mm,	Y =  169.000  mm,	Z =   -1.000 mm,
	W =-180.000 deg,	P =   0.000 deg,	R =    90.000 deg
};
P[7881]{
   GP1:
	UF : 1, UT : 4,		CONFIG : 'N U T, 0, 0, 0',
	X =  112.000  mm,	Y =  169.000  mm,	Z =   15.000 mm,
	W =-180.000 deg,	P =   0.000 deg,	R =    90.000 deg
};
P[7885]{
   GP1:
	UF : 1, UT : 4,		CONFIG : 'N U T, 0, 0, 0',
	X =  118.000  mm,	Y =  169.000  mm,	Z =   15.000 mm,
	W =-180.000 deg,	P =   0.000 deg,	R =    90.000 deg
};
P[7886]{
   GP1:
	UF : 1, UT : 4,		CONFIG : 'N U T, 0, 0, 0',
	X =  118.000  mm,	Y =  169.000  mm,	Z =   -1.000 mm,
	W =-180.000 deg,	P =   0.000 deg,	R =    90.000 deg
};
P[7887]{
   GP1:
	UF : 1, UT : 4,		CONFIG : 'N U T, 0, 0, 0',
	X =  118.000  mm,	Y =  169.000  mm,	Z =   15.000 mm,
	W =-180.000 deg,	P =   0.000 deg,	R =    90.000 deg
};
P[7894]{
   GP1:
	UF : 1, UT : 4,		CONFIG : 'N U T, 0, 0, 0',
	X =  127.000  mm,	Y =  169.000  mm,	Z =   15.000 mm,
	W =-180.000 deg,	P =   0.000 deg,	R =    90.000 deg
};
P[7895]{
   GP1:
	UF : 1, UT : 4,		CONFIG : 'N U T, 0, 0, 0',
	X =  127.000  mm,	Y =  169.000  mm,	Z =   -1.000 mm,
	W =-180.000 deg,	P =   0.000 deg,	R =    90.000 deg
};
P[7896]{
   GP1:
	UF : 1, UT : 4,		CONFIG : 'N U T, 0, 0, 0',
	X =  127.000  mm,	Y =  169.000  mm,	Z =   15.000 mm,
	W =-180.000 deg,	P =   0.000 deg,	R =    90.000 deg
};
P[7897]{
   GP1:
	UF : 1, UT : 4,		CONFIG : 'N U T, 0, 0, 0',
	X =  130.000  mm,	Y =  169.000  mm,	Z =   15.000 mm,
	W =-180.000 deg,	P =   0.000 deg,	R =    90.000 deg
};
P[7898]{
   GP1:
	UF : 1, UT : 4,		CONFIG : 'N U T, 0, 0, 0',
	X =  130.000  mm,	Y =  169.000  mm,	Z =   -1.000 mm,
	W =-180.000 deg,	P =   0.000 deg,	R =    90.000 deg
};
P[7899]{
   GP1:
	UF : 1, UT : 4,		CONFIG : 'N U T, 0, 0, 0',
	X =  130.000  mm,	Y =  169.000  mm,	Z =   15.000 mm,
	W =-180.000 deg,	P =   0.000 deg,	R =    90.000 deg
};
P[7903]{
   GP1:
	UF : 1, UT : 4,		CONFIG : 'N U T, 0, 0, 0',
	X =  136.000  mm,	Y =  169.000  mm,	Z =   15.000 mm,
	W =-180.000 deg,	P =   0.000 deg,	R =    90.000 deg
};
P[7904]{
   GP1:
	UF : 1, UT : 4,		CONFIG : 'N U T, 0, 0, 0',
	X =  136.000  mm,	Y =  169.000  mm,	Z =   -1.000 mm,
	W =-180.000 deg,	P =   0.000 deg,	R =    90.000 deg
};
P[7905]{
   GP1:
	UF : 1, UT : 4,		CONFIG : 'N U T, 0, 0, 0',
	X =  136.000  mm,	Y =  169.000  mm,	Z =   15.000 mm,
	W =-180.000 deg,	P =   0.000 deg,	R =    90.000 deg
};
P[7906]{
   GP1:
	UF : 1, UT : 4,		CONFIG : 'N U T, 0, 0, 0',
	X =  139.000  mm,	Y =  169.000  mm,	Z =   15.000 mm,
	W =-180.000 deg,	P =   0.000 deg,	R =    90.000 deg
};
P[7907]{
   GP1:
	UF : 1, UT : 4,		CONFIG : 'N U T, 0, 0, 0',
	X =  139.000  mm,	Y =  169.000  mm,	Z =   -1.000 mm,
	W =-180.000 deg,	P =   0.000 deg,	R =    90.000 deg
};
P[7908]{
   GP1:
	UF : 1, UT : 4,		CONFIG : 'N U T, 0, 0, 0',
	X =  139.000  mm,	Y =  169.000  mm,	Z =   15.000 mm,
	W =-180.000 deg,	P =   0.000 deg,	R =    90.000 deg
};
P[7909]{
   GP1:
	UF : 1, UT : 4,		CONFIG : 'N U T, 0, 0, 0',
	X =  142.000  mm,	Y =  169.000  mm,	Z =   15.000 mm,
	W =-180.000 deg,	P =   0.000 deg,	R =    90.000 deg
};
P[7910]{
   GP1:
	UF : 1, UT : 4,		CONFIG : 'N U T, 0, 0, 0',
	X =  142.000  mm,	Y =  169.000  mm,	Z =   -1.000 mm,
	W =-180.000 deg,	P =   0.000 deg,	R =    90.000 deg
};
P[7911]{
   GP1:
	UF : 1, UT : 4,		CONFIG : 'N U T, 0, 0, 0',
	X =  142.000  mm,	Y =  169.000  mm,	Z =   15.000 mm,
	W =-180.000 deg,	P =   0.000 deg,	R =    90.000 deg
};
P[7912]{
   GP1:
	UF : 1, UT : 4,		CONFIG : 'N U T, 0, 0, 0',
	X =  145.000  mm,	Y =  169.000  mm,	Z =   15.000 mm,
	W =-180.000 deg,	P =   0.000 deg,	R =    90.000 deg
};
P[7913]{
   GP1:
	UF : 1, UT : 4,		CONFIG : 'N U T, 0, 0, 0',
	X =  145.000  mm,	Y =  169.000  mm,	Z =   -1.000 mm,
	W =-180.000 deg,	P =   0.000 deg,	R =    90.000 deg
};
P[7914]{
   GP1:
	UF : 1, UT : 4,		CONFIG : 'N U T, 0, 0, 0',
	X =  145.000  mm,	Y =  169.000  mm,	Z =   15.000 mm,
	W =-180.000 deg,	P =   0.000 deg,	R =    90.000 deg
};
P[7915]{
   GP1:
	UF : 1, UT : 4,		CONFIG : 'N U T, 0, 0, 0',
	X =  148.000  mm,	Y =  169.000  mm,	Z =   15.000 mm,
	W =-180.000 deg,	P =   0.000 deg,	R =    90.000 deg
};
P[7916]{
   GP1:
	UF : 1, UT : 4,		CONFIG : 'N U T, 0, 0, 0',
	X =  148.000  mm,	Y =  169.000  mm,	Z =   -1.000 mm,
	W =-180.000 deg,	P =   0.000 deg,	R =    90.000 deg
};
P[7917]{
   GP1:
	UF : 1, UT : 4,		CONFIG : 'N U T, 0, 0, 0',
	X =  148.000  mm,	Y =  169.000  mm,	Z =   15.000 mm,
	W =-180.000 deg,	P =   0.000 deg,	R =    90.000 deg
};
P[7921]{
   GP1:
	UF : 1, UT : 4,		CONFIG : 'N U T, 0, 0, 0',
	X =  154.000  mm,	Y =  169.000  mm,	Z =   15.000 mm,
	W =-180.000 deg,	P =   0.000 deg,	R =    90.000 deg
};
P[7922]{
   GP1:
	UF : 1, UT : 4,		CONFIG : 'N U T, 0, 0, 0',
	X =  154.000  mm,	Y =  169.000  mm,	Z =   -1.000 mm,
	W =-180.000 deg,	P =   0.000 deg,	R =    90.000 deg
};
P[7923]{
   GP1:
	UF : 1, UT : 4,		CONFIG : 'N U T, 0, 0, 0',
	X =  154.000  mm,	Y =  169.000  mm,	Z =   15.000 mm,
	W =-180.000 deg,	P =   0.000 deg,	R =    90.000 deg
};
P[7924]{
   GP1:
	UF : 1, UT : 4,		CONFIG : 'N U T, 0, 0, 0',
	X =  31.000  mm,	Y =  172.000  mm,	Z =   15.000 mm,
	W =-180.000 deg,	P =   0.000 deg,	R =    90.000 deg
};
P[7925]{
   GP1:
	UF : 1, UT : 4,		CONFIG : 'N U T, 0, 0, 0',
	X =  31.000  mm,	Y =  172.000  mm,	Z =   -1.000 mm,
	W =-180.000 deg,	P =   0.000 deg,	R =    90.000 deg
};
P[7926]{
   GP1:
	UF : 1, UT : 4,		CONFIG : 'N U T, 0, 0, 0',
	X =  31.000  mm,	Y =  172.000  mm,	Z =   15.000 mm,
	W =-180.000 deg,	P =   0.000 deg,	R =    90.000 deg
};
P[7933]{
   GP1:
	UF : 1, UT : 4,		CONFIG : 'N U T, 0, 0, 0',
	X =  43.000  mm,	Y =  172.000  mm,	Z =   15.000 mm,
	W =-180.000 deg,	P =   0.000 deg,	R =    90.000 deg
};
P[7934]{
   GP1:
	UF : 1, UT : 4,		CONFIG : 'N U T, 0, 0, 0',
	X =  43.000  mm,	Y =  172.000  mm,	Z =   -1.000 mm,
	W =-180.000 deg,	P =   0.000 deg,	R =    90.000 deg
};
P[7935]{
   GP1:
	UF : 1, UT : 4,		CONFIG : 'N U T, 0, 0, 0',
	X =  43.000  mm,	Y =  172.000  mm,	Z =   15.000 mm,
	W =-180.000 deg,	P =   0.000 deg,	R =    90.000 deg
};
P[7966]{
   GP1:
	UF : 1, UT : 4,		CONFIG : 'N U T, 0, 0, 0',
	X =  127.000  mm,	Y =  172.000  mm,	Z =   15.000 mm,
	W =-180.000 deg,	P =   0.000 deg,	R =    90.000 deg
};
P[7967]{
   GP1:
	UF : 1, UT : 4,		CONFIG : 'N U T, 0, 0, 0',
	X =  127.000  mm,	Y =  172.000  mm,	Z =   -1.000 mm,
	W =-180.000 deg,	P =   0.000 deg,	R =    90.000 deg
};
P[7968]{
   GP1:
	UF : 1, UT : 4,		CONFIG : 'N U T, 0, 0, 0',
	X =  127.000  mm,	Y =  172.000  mm,	Z =   15.000 mm,
	W =-180.000 deg,	P =   0.000 deg,	R =    90.000 deg
};
P[7969]{
   GP1:
	UF : 1, UT : 4,		CONFIG : 'N U T, 0, 0, 0',
	X =  130.000  mm,	Y =  172.000  mm,	Z =   15.000 mm,
	W =-180.000 deg,	P =   0.000 deg,	R =    90.000 deg
};
P[7970]{
   GP1:
	UF : 1, UT : 4,		CONFIG : 'N U T, 0, 0, 0',
	X =  130.000  mm,	Y =  172.000  mm,	Z =   -1.000 mm,
	W =-180.000 deg,	P =   0.000 deg,	R =    90.000 deg
};
P[7971]{
   GP1:
	UF : 1, UT : 4,		CONFIG : 'N U T, 0, 0, 0',
	X =  130.000  mm,	Y =  172.000  mm,	Z =   15.000 mm,
	W =-180.000 deg,	P =   0.000 deg,	R =    90.000 deg
};
P[7972]{
   GP1:
	UF : 1, UT : 4,		CONFIG : 'N U T, 0, 0, 0',
	X =  133.000  mm,	Y =  172.000  mm,	Z =   15.000 mm,
	W =-180.000 deg,	P =   0.000 deg,	R =    90.000 deg
};
P[7973]{
   GP1:
	UF : 1, UT : 4,		CONFIG : 'N U T, 0, 0, 0',
	X =  133.000  mm,	Y =  172.000  mm,	Z =   -1.000 mm,
	W =-180.000 deg,	P =   0.000 deg,	R =    90.000 deg
};
P[7974]{
   GP1:
	UF : 1, UT : 4,		CONFIG : 'N U T, 0, 0, 0',
	X =  133.000  mm,	Y =  172.000  mm,	Z =   15.000 mm,
	W =-180.000 deg,	P =   0.000 deg,	R =    90.000 deg
};
P[7975]{
   GP1:
	UF : 1, UT : 4,		CONFIG : 'N U T, 0, 0, 0',
	X =  136.000  mm,	Y =  172.000  mm,	Z =   15.000 mm,
	W =-180.000 deg,	P =   0.000 deg,	R =    90.000 deg
};
P[7976]{
   GP1:
	UF : 1, UT : 4,		CONFIG : 'N U T, 0, 0, 0',
	X =  136.000  mm,	Y =  172.000  mm,	Z =   -1.000 mm,
	W =-180.000 deg,	P =   0.000 deg,	R =    90.000 deg
};
P[7977]{
   GP1:
	UF : 1, UT : 4,		CONFIG : 'N U T, 0, 0, 0',
	X =  136.000  mm,	Y =  172.000  mm,	Z =   15.000 mm,
	W =-180.000 deg,	P =   0.000 deg,	R =    90.000 deg
};
P[7978]{
   GP1:
	UF : 1, UT : 4,		CONFIG : 'N U T, 0, 0, 0',
	X =  139.000  mm,	Y =  172.000  mm,	Z =   15.000 mm,
	W =-180.000 deg,	P =   0.000 deg,	R =    90.000 deg
};
P[7979]{
   GP1:
	UF : 1, UT : 4,		CONFIG : 'N U T, 0, 0, 0',
	X =  139.000  mm,	Y =  172.000  mm,	Z =   -1.000 mm,
	W =-180.000 deg,	P =   0.000 deg,	R =    90.000 deg
};
P[7980]{
   GP1:
	UF : 1, UT : 4,		CONFIG : 'N U T, 0, 0, 0',
	X =  139.000  mm,	Y =  172.000  mm,	Z =   15.000 mm,
	W =-180.000 deg,	P =   0.000 deg,	R =    90.000 deg
};
P[7981]{
   GP1:
	UF : 1, UT : 4,		CONFIG : 'N U T, 0, 0, 0',
	X =  142.000  mm,	Y =  172.000  mm,	Z =   15.000 mm,
	W =-180.000 deg,	P =   0.000 deg,	R =    90.000 deg
};
P[7982]{
   GP1:
	UF : 1, UT : 4,		CONFIG : 'N U T, 0, 0, 0',
	X =  142.000  mm,	Y =  172.000  mm,	Z =   -1.000 mm,
	W =-180.000 deg,	P =   0.000 deg,	R =    90.000 deg
};
P[7983]{
   GP1:
	UF : 1, UT : 4,		CONFIG : 'N U T, 0, 0, 0',
	X =  142.000  mm,	Y =  172.000  mm,	Z =   15.000 mm,
	W =-180.000 deg,	P =   0.000 deg,	R =    90.000 deg
};
P[7984]{
   GP1:
	UF : 1, UT : 4,		CONFIG : 'N U T, 0, 0, 0',
	X =  145.000  mm,	Y =  172.000  mm,	Z =   15.000 mm,
	W =-180.000 deg,	P =   0.000 deg,	R =    90.000 deg
};
P[7985]{
   GP1:
	UF : 1, UT : 4,		CONFIG : 'N U T, 0, 0, 0',
	X =  145.000  mm,	Y =  172.000  mm,	Z =   -1.000 mm,
	W =-180.000 deg,	P =   0.000 deg,	R =    90.000 deg
};
P[7986]{
   GP1:
	UF : 1, UT : 4,		CONFIG : 'N U T, 0, 0, 0',
	X =  145.000  mm,	Y =  172.000  mm,	Z =   15.000 mm,
	W =-180.000 deg,	P =   0.000 deg,	R =    90.000 deg
};
P[7993]{
   GP1:
	UF : 1, UT : 4,		CONFIG : 'N U T, 0, 0, 0',
	X =  1.000  mm,	Y =  175.000  mm,	Z =   15.000 mm,
	W =-180.000 deg,	P =   0.000 deg,	R =    90.000 deg
};
P[7994]{
   GP1:
	UF : 1, UT : 4,		CONFIG : 'N U T, 0, 0, 0',
	X =  1.000  mm,	Y =  175.000  mm,	Z =   -1.000 mm,
	W =-180.000 deg,	P =   0.000 deg,	R =    90.000 deg
};
P[7995]{
   GP1:
	UF : 1, UT : 4,		CONFIG : 'N U T, 0, 0, 0',
	X =  1.000  mm,	Y =  175.000  mm,	Z =   15.000 mm,
	W =-180.000 deg,	P =   0.000 deg,	R =    90.000 deg
};
P[8008]{
   GP1:
	UF : 1, UT : 4,		CONFIG : 'N U T, 0, 0, 0',
	X =  106.000  mm,	Y =  175.000  mm,	Z =   15.000 mm,
	W =-180.000 deg,	P =   0.000 deg,	R =    90.000 deg
};
P[8009]{
   GP1:
	UF : 1, UT : 4,		CONFIG : 'N U T, 0, 0, 0',
	X =  106.000  mm,	Y =  175.000  mm,	Z =   -1.000 mm,
	W =-180.000 deg,	P =   0.000 deg,	R =    90.000 deg
};
P[8010]{
   GP1:
	UF : 1, UT : 4,		CONFIG : 'N U T, 0, 0, 0',
	X =  106.000  mm,	Y =  175.000  mm,	Z =   15.000 mm,
	W =-180.000 deg,	P =   0.000 deg,	R =    90.000 deg
};
P[8035]{
   GP1:
	UF : 1, UT : 4,		CONFIG : 'N U T, 0, 0, 0',
	X =  133.000  mm,	Y =  175.000  mm,	Z =   15.000 mm,
	W =-180.000 deg,	P =   0.000 deg,	R =    90.000 deg
};
P[8036]{
   GP1:
	UF : 1, UT : 4,		CONFIG : 'N U T, 0, 0, 0',
	X =  133.000  mm,	Y =  175.000  mm,	Z =   -1.000 mm,
	W =-180.000 deg,	P =   0.000 deg,	R =    90.000 deg
};
P[8037]{
   GP1:
	UF : 1, UT : 4,		CONFIG : 'N U T, 0, 0, 0',
	X =  133.000  mm,	Y =  175.000  mm,	Z =   15.000 mm,
	W =-180.000 deg,	P =   0.000 deg,	R =    90.000 deg
};
P[8038]{
   GP1:
	UF : 1, UT : 4,		CONFIG : 'N U T, 0, 0, 0',
	X =  136.000  mm,	Y =  175.000  mm,	Z =   15.000 mm,
	W =-180.000 deg,	P =   0.000 deg,	R =    90.000 deg
};
P[8039]{
   GP1:
	UF : 1, UT : 4,		CONFIG : 'N U T, 0, 0, 0',
	X =  136.000  mm,	Y =  175.000  mm,	Z =   -1.000 mm,
	W =-180.000 deg,	P =   0.000 deg,	R =    90.000 deg
};
P[8040]{
   GP1:
	UF : 1, UT : 4,		CONFIG : 'N U T, 0, 0, 0',
	X =  136.000  mm,	Y =  175.000  mm,	Z =   15.000 mm,
	W =-180.000 deg,	P =   0.000 deg,	R =    90.000 deg
};
P[8041]{
   GP1:
	UF : 1, UT : 4,		CONFIG : 'N U T, 0, 0, 0',
	X =  139.000  mm,	Y =  175.000  mm,	Z =   15.000 mm,
	W =-180.000 deg,	P =   0.000 deg,	R =    90.000 deg
};
P[8042]{
   GP1:
	UF : 1, UT : 4,		CONFIG : 'N U T, 0, 0, 0',
	X =  139.000  mm,	Y =  175.000  mm,	Z =   -1.000 mm,
	W =-180.000 deg,	P =   0.000 deg,	R =    90.000 deg
};
P[8043]{
   GP1:
	UF : 1, UT : 4,		CONFIG : 'N U T, 0, 0, 0',
	X =  139.000  mm,	Y =  175.000  mm,	Z =   15.000 mm,
	W =-180.000 deg,	P =   0.000 deg,	R =    90.000 deg
};
P[8044]{
   GP1:
	UF : 1, UT : 4,		CONFIG : 'N U T, 0, 0, 0',
	X =  142.000  mm,	Y =  175.000  mm,	Z =   15.000 mm,
	W =-180.000 deg,	P =   0.000 deg,	R =    90.000 deg
};
P[8045]{
   GP1:
	UF : 1, UT : 4,		CONFIG : 'N U T, 0, 0, 0',
	X =  142.000  mm,	Y =  175.000  mm,	Z =   -1.000 mm,
	W =-180.000 deg,	P =   0.000 deg,	R =    90.000 deg
};
P[8046]{
   GP1:
	UF : 1, UT : 4,		CONFIG : 'N U T, 0, 0, 0',
	X =  142.000  mm,	Y =  175.000  mm,	Z =   15.000 mm,
	W =-180.000 deg,	P =   0.000 deg,	R =    90.000 deg
};
P[8068]{
   GP1:
	UF : 1, UT : 4,		CONFIG : 'N U T, 0, 0, 0',
	X =  16.000  mm,	Y =  178.000  mm,	Z =   15.000 mm,
	W =-180.000 deg,	P =   0.000 deg,	R =    90.000 deg
};
P[8069]{
   GP1:
	UF : 1, UT : 4,		CONFIG : 'N U T, 0, 0, 0',
	X =  16.000  mm,	Y =  178.000  mm,	Z =   -1.000 mm,
	W =-180.000 deg,	P =   0.000 deg,	R =    90.000 deg
};
P[8070]{
   GP1:
	UF : 1, UT : 4,		CONFIG : 'N U T, 0, 0, 0',
	X =  16.000  mm,	Y =  178.000  mm,	Z =   15.000 mm,
	W =-180.000 deg,	P =   0.000 deg,	R =    90.000 deg
};
P[8071]{
   GP1:
	UF : 1, UT : 4,		CONFIG : 'N U T, 0, 0, 0',
	X =  19.000  mm,	Y =  178.000  mm,	Z =   15.000 mm,
	W =-180.000 deg,	P =   0.000 deg,	R =    90.000 deg
};
P[8072]{
   GP1:
	UF : 1, UT : 4,		CONFIG : 'N U T, 0, 0, 0',
	X =  19.000  mm,	Y =  178.000  mm,	Z =   -1.000 mm,
	W =-180.000 deg,	P =   0.000 deg,	R =    90.000 deg
};
P[8073]{
   GP1:
	UF : 1, UT : 4,		CONFIG : 'N U T, 0, 0, 0',
	X =  19.000  mm,	Y =  178.000  mm,	Z =   15.000 mm,
	W =-180.000 deg,	P =   0.000 deg,	R =    90.000 deg
};
P[8116]{
   GP1:
	UF : 1, UT : 4,		CONFIG : 'N U T, 0, 0, 0',
	X =  151.000  mm,	Y =  178.000  mm,	Z =   15.000 mm,
	W =-180.000 deg,	P =   0.000 deg,	R =    90.000 deg
};
P[8117]{
   GP1:
	UF : 1, UT : 4,		CONFIG : 'N U T, 0, 0, 0',
	X =  151.000  mm,	Y =  178.000  mm,	Z =   -1.000 mm,
	W =-180.000 deg,	P =   0.000 deg,	R =    90.000 deg
};
P[8118]{
   GP1:
	UF : 1, UT : 4,		CONFIG : 'N U T, 0, 0, 0',
	X =  151.000  mm,	Y =  178.000  mm,	Z =   15.000 mm,
	W =-180.000 deg,	P =   0.000 deg,	R =    90.000 deg
};
P[8149]{
   GP1:
	UF : 1, UT : 4,		CONFIG : 'N U T, 0, 0, 0',
	X =  16.000  mm,	Y =  181.000  mm,	Z =   15.000 mm,
	W =-180.000 deg,	P =   0.000 deg,	R =    90.000 deg
};
P[8150]{
   GP1:
	UF : 1, UT : 4,		CONFIG : 'N U T, 0, 0, 0',
	X =  16.000  mm,	Y =  181.000  mm,	Z =   -1.000 mm,
	W =-180.000 deg,	P =   0.000 deg,	R =    90.000 deg
};
P[8151]{
   GP1:
	UF : 1, UT : 4,		CONFIG : 'N U T, 0, 0, 0',
	X =  16.000  mm,	Y =  181.000  mm,	Z =   15.000 mm,
	W =-180.000 deg,	P =   0.000 deg,	R =    90.000 deg
};
P[8158]{
   GP1:
	UF : 1, UT : 4,		CONFIG : 'N U T, 0, 0, 0',
	X =  109.000  mm,	Y =  181.000  mm,	Z =   15.000 mm,
	W =-180.000 deg,	P =   0.000 deg,	R =    90.000 deg
};
P[8159]{
   GP1:
	UF : 1, UT : 4,		CONFIG : 'N U T, 0, 0, 0',
	X =  109.000  mm,	Y =  181.000  mm,	Z =   -1.000 mm,
	W =-180.000 deg,	P =   0.000 deg,	R =    90.000 deg
};
P[8160]{
   GP1:
	UF : 1, UT : 4,		CONFIG : 'N U T, 0, 0, 0',
	X =  109.000  mm,	Y =  181.000  mm,	Z =   15.000 mm,
	W =-180.000 deg,	P =   0.000 deg,	R =    90.000 deg
};
P[8164]{
   GP1:
	UF : 1, UT : 4,		CONFIG : 'N U T, 0, 0, 0',
	X =  115.000  mm,	Y =  181.000  mm,	Z =   15.000 mm,
	W =-180.000 deg,	P =   0.000 deg,	R =    90.000 deg
};
P[8165]{
   GP1:
	UF : 1, UT : 4,		CONFIG : 'N U T, 0, 0, 0',
	X =  115.000  mm,	Y =  181.000  mm,	Z =   -1.000 mm,
	W =-180.000 deg,	P =   0.000 deg,	R =    90.000 deg
};
P[8166]{
   GP1:
	UF : 1, UT : 4,		CONFIG : 'N U T, 0, 0, 0',
	X =  115.000  mm,	Y =  181.000  mm,	Z =   15.000 mm,
	W =-180.000 deg,	P =   0.000 deg,	R =    90.000 deg
};
P[8170]{
   GP1:
	UF : 1, UT : 4,		CONFIG : 'N U T, 0, 0, 0',
	X =  121.000  mm,	Y =  181.000  mm,	Z =   15.000 mm,
	W =-180.000 deg,	P =   0.000 deg,	R =    90.000 deg
};
P[8171]{
   GP1:
	UF : 1, UT : 4,		CONFIG : 'N U T, 0, 0, 0',
	X =  121.000  mm,	Y =  181.000  mm,	Z =   -1.000 mm,
	W =-180.000 deg,	P =   0.000 deg,	R =    90.000 deg
};
P[8172]{
   GP1:
	UF : 1, UT : 4,		CONFIG : 'N U T, 0, 0, 0',
	X =  121.000  mm,	Y =  181.000  mm,	Z =   15.000 mm,
	W =-180.000 deg,	P =   0.000 deg,	R =    90.000 deg
};
P[8191]{
   GP1:
	UF : 1, UT : 4,		CONFIG : 'N U T, 0, 0, 0',
	X =  142.000  mm,	Y =  181.000  mm,	Z =   15.000 mm,
	W =-180.000 deg,	P =   0.000 deg,	R =    90.000 deg
};
P[8192]{
   GP1:
	UF : 1, UT : 4,		CONFIG : 'N U T, 0, 0, 0',
	X =  142.000  mm,	Y =  181.000  mm,	Z =   -1.000 mm,
	W =-180.000 deg,	P =   0.000 deg,	R =    90.000 deg
};
P[8193]{
   GP1:
	UF : 1, UT : 4,		CONFIG : 'N U T, 0, 0, 0',
	X =  142.000  mm,	Y =  181.000  mm,	Z =   15.000 mm,
	W =-180.000 deg,	P =   0.000 deg,	R =    90.000 deg
};
P[8260]{
   GP1:
	UF : 1, UT : 4,		CONFIG : 'N U T, 0, 0, 0',
	X =  31.000  mm,	Y =  184.000  mm,	Z =   15.000 mm,
	W =-180.000 deg,	P =   0.000 deg,	R =    90.000 deg
};
P[8261]{
   GP1:
	UF : 1, UT : 4,		CONFIG : 'N U T, 0, 0, 0',
	X =  31.000  mm,	Y =  184.000  mm,	Z =   -1.000 mm,
	W =-180.000 deg,	P =   0.000 deg,	R =    90.000 deg
};
P[8262]{
   GP1:
	UF : 1, UT : 4,		CONFIG : 'N U T, 0, 0, 0',
	X =  31.000  mm,	Y =  184.000  mm,	Z =   15.000 mm,
	W =-180.000 deg,	P =   0.000 deg,	R =    90.000 deg
};
P[8263]{
   GP1:
	UF : 1, UT : 4,		CONFIG : 'N U T, 0, 0, 0',
	X =  112.000  mm,	Y =  184.000  mm,	Z =   15.000 mm,
	W =-180.000 deg,	P =   0.000 deg,	R =    90.000 deg
};
P[8264]{
   GP1:
	UF : 1, UT : 4,		CONFIG : 'N U T, 0, 0, 0',
	X =  112.000  mm,	Y =  184.000  mm,	Z =   -1.000 mm,
	W =-180.000 deg,	P =   0.000 deg,	R =    90.000 deg
};
P[8265]{
   GP1:
	UF : 1, UT : 4,		CONFIG : 'N U T, 0, 0, 0',
	X =  112.000  mm,	Y =  184.000  mm,	Z =   15.000 mm,
	W =-180.000 deg,	P =   0.000 deg,	R =    90.000 deg
};
P[8266]{
   GP1:
	UF : 1, UT : 4,		CONFIG : 'N U T, 0, 0, 0',
	X =  115.000  mm,	Y =  184.000  mm,	Z =   15.000 mm,
	W =-180.000 deg,	P =   0.000 deg,	R =    90.000 deg
};
P[8267]{
   GP1:
	UF : 1, UT : 4,		CONFIG : 'N U T, 0, 0, 0',
	X =  115.000  mm,	Y =  184.000  mm,	Z =   -1.000 mm,
	W =-180.000 deg,	P =   0.000 deg,	R =    90.000 deg
};
P[8268]{
   GP1:
	UF : 1, UT : 4,		CONFIG : 'N U T, 0, 0, 0',
	X =  115.000  mm,	Y =  184.000  mm,	Z =   15.000 mm,
	W =-180.000 deg,	P =   0.000 deg,	R =    90.000 deg
};
P[8293]{
   GP1:
	UF : 1, UT : 4,		CONFIG : 'N U T, 0, 0, 0',
	X =  142.000  mm,	Y =  184.000  mm,	Z =   15.000 mm,
	W =-180.000 deg,	P =   0.000 deg,	R =    90.000 deg
};
P[8294]{
   GP1:
	UF : 1, UT : 4,		CONFIG : 'N U T, 0, 0, 0',
	X =  142.000  mm,	Y =  184.000  mm,	Z =   -1.000 mm,
	W =-180.000 deg,	P =   0.000 deg,	R =    90.000 deg
};
P[8295]{
   GP1:
	UF : 1, UT : 4,		CONFIG : 'N U T, 0, 0, 0',
	X =  142.000  mm,	Y =  184.000  mm,	Z =   15.000 mm,
	W =-180.000 deg,	P =   0.000 deg,	R =    90.000 deg
};
P[8449]{
   GP1:
	UF : 1, UT : 4,		CONFIG : 'N U T, 0, 0, 0',
	X =  121.000  mm,	Y =  187.000  mm,	Z =   15.000 mm,
	W =-180.000 deg,	P =   0.000 deg,	R =    90.000 deg
};
P[8450]{
   GP1:
	UF : 1, UT : 4,		CONFIG : 'N U T, 0, 0, 0',
	X =  121.000  mm,	Y =  187.000  mm,	Z =   -1.000 mm,
	W =-180.000 deg,	P =   0.000 deg,	R =    90.000 deg
};
P[8451]{
   GP1:
	UF : 1, UT : 4,		CONFIG : 'N U T, 0, 0, 0',
	X =  121.000  mm,	Y =  187.000  mm,	Z =   15.000 mm,
	W =-180.000 deg,	P =   0.000 deg,	R =    90.000 deg
};
P[11569]{
   GP1:
	UF : 1, UT : 4,		CONFIG : 'N U T, 0, 0, 0',
	X =  145.000  mm,	Y =  300.000  mm,	Z =   100.000 mm,
	W =-180.000 deg,	P =   0.000 deg,	R =    90.000 deg
};
/END
